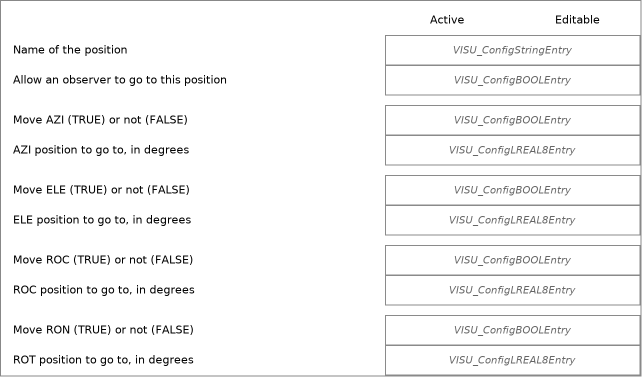
VISUALIZATION VISU_AxesConfig_KnownPosition  // 642x377
VAR_IN_OUT
    editable : AxesKnownPositionConfig;
	active : AxesKnownPositionConfig;
END_VAR
    Frame (385,35 255x30)
        shows VISU_ConfigStringEntry(active := active.name, editable := editable.name)
    Label (385,10 125x20), "Active"
    Label (515,10 125x20), "Editable"
    Label (10,35 370x30), "Name of the position"
    Frame (385,65 255x30)
        shows VISU_ConfigBOOLEntry(active := active.allowObserver, editable := editable.allowObserver)
    Label (10,65 370x30), "Allow an observer to go to this position"
    Label (10,135 370x30), "AZI position to go to, in degrees"
    Frame (385,135 255x30)
        shows VISU_ConfigLREAL8Entry(active := active.azi, editable := editable.azi)
    Label (10,105 370x30), "Move AZI (TRUE) or not (FALSE)"
    Frame (385,105 255x30)
        shows VISU_ConfigBOOLEntry(active := active.doAzi, editable := editable.doAzi)
    Label (10,205 370x30), "ELE position to go to, in degrees"
    Frame (385,205 255x30)
        shows VISU_ConfigLREAL8Entry(active := active.ele, editable := editable.ele)
    Label (10,175 370x30), "Move ELE (TRUE) or not (FALSE)"
    Frame (385,175 255x30)
        shows VISU_ConfigBOOLEntry(active := active.doEle, editable := editable.doEle)
    Label (10,275 370x30), "ROC position to go to, in degrees"
    Frame (385,275 255x30)
        shows VISU_ConfigLREAL8Entry(active := active.roc, editable := editable.roc)
    Label (10,245 370x30), "Move ROC (TRUE) or not (FALSE)"
    Frame (385,245 255x30)
        shows VISU_ConfigBOOLEntry(active := active.doRoc, editable := editable.doRoc)
    Label (10,345 370x30), "ROT position to go to, in degrees"
    Frame (385,345 255x30)
        shows VISU_ConfigLREAL8Entry(active := active.ron, editable := editable.ron)
    Label (10,315 370x30), "Move RON (TRUE) or not (FALSE)"
    Frame (385,315 255x30)
        shows VISU_ConfigBOOLEntry(active := active.doRon, editable := editable.doRon)
END_VISUALIZATION

(* stored: Version 1.1.0.1, ProductVersion 3.1.4019.2
   Visu VISU_AxesConfig_KnownPosition: Id {93c046ca-3f16-4eda-99ec-fc4240d95434} *)
